VAR_GLOBAL PERSISTENT
	
	aDataHistory					: ARRAY [0..200] OF ST_CycleData;
	nIndexDataHistory				: DINT;	

/////////////////////////////////////////////////////////////////////////////////////Event Log/////////////////////////////////////////////////////////////////////////////////////
	
	stAlarmHistory				: ARRAY [00..250] OF ST_AlarmHistory;
	aEventLog					: ARRAY [0..250] OF T_MaxSTring;	//Event log - connected to alarm history in HMI	
	aTimeLog					: ARRAY [0..250] OF T_MaxSTring;
	aDateLog					: ARRAY [0..250] OF T_MaxSTring;	
	
	stUserLog					: ARRAY [0..250] OF ST_UserLog;
	
	stStatisticsHMI				: ARRAY [0..3] OF ST_StatisticsHMI;	//0: GENERAL
																	//1: STATION 1
																	//2: STATION 2
																	//3: STATION 3
	


END_VAR

(* stored: Version 1.1.0.1, ProductVersion 3.1.4024.13
   GVL GVL_Persistent: Id {c4d03ea6-35af-4633-972d-fef3cfe7daa9} *)
